{attribute 'qualified_only'}
VAR_GLOBAL
	THT : ARRAY [1..14] OF RTU_THT;
END_VAR


VAR_GLOBAL CONSTANT
	Temp_OOR_Min : REAL :=   0.0;
	Temp_OOR_Max : REAL :=  50.0;
	RH_OOR_Min   : REAL :=   0.0;
	RH_OOR_Max   : REAL := 100.0;
END_VAR

(* stored: Version 1.1.0.1, ProductVersion 3.1.4024.12
   GVL GVL_THT: Id {052ef35f-7cf7-4131-bd38-b8b866382700} *)
